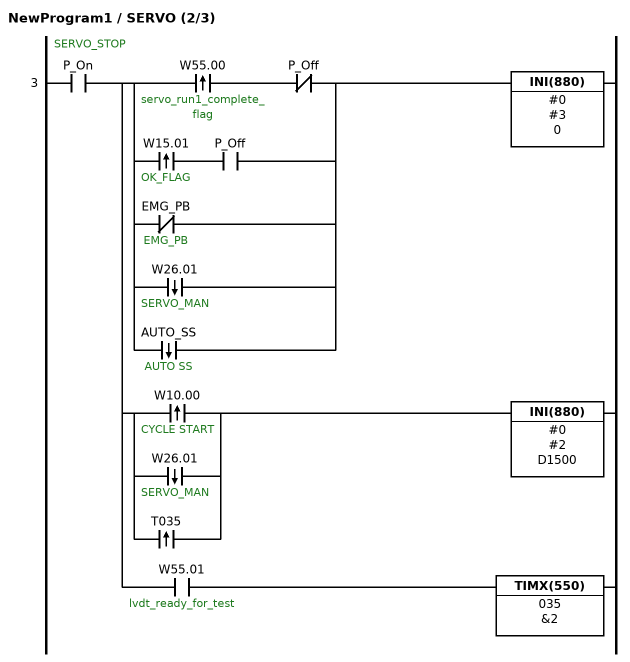
; [picture p24: NewProgram1 / SERVO, rungs 3-3]
; rung 3: SERVO_STOP
LD P_On
OUT TR0
@LD W55.00  ; servo_run1_complete_flag
ANDNOT P_Off
@LD W15.01  ; OK_FLAG
AND P_Off
ORLD
ORNOT EMG_PB  ; EMG_PB
%OR W26.01  ; SERVO_MAN
%OR AUTO_SS  ; AUTO SS
ANDLD
INI(880) #0 #3 0
LD TR0
@LD W10.00  ; CYCLE START
%OR W26.01  ; SERVO_MAN
@OR T035
ANDLD
INI(880) #0 #2 D1500
LD TR0
AND W55.01  ; lvdt_ready_for_test
TIMX(550) 035 &2

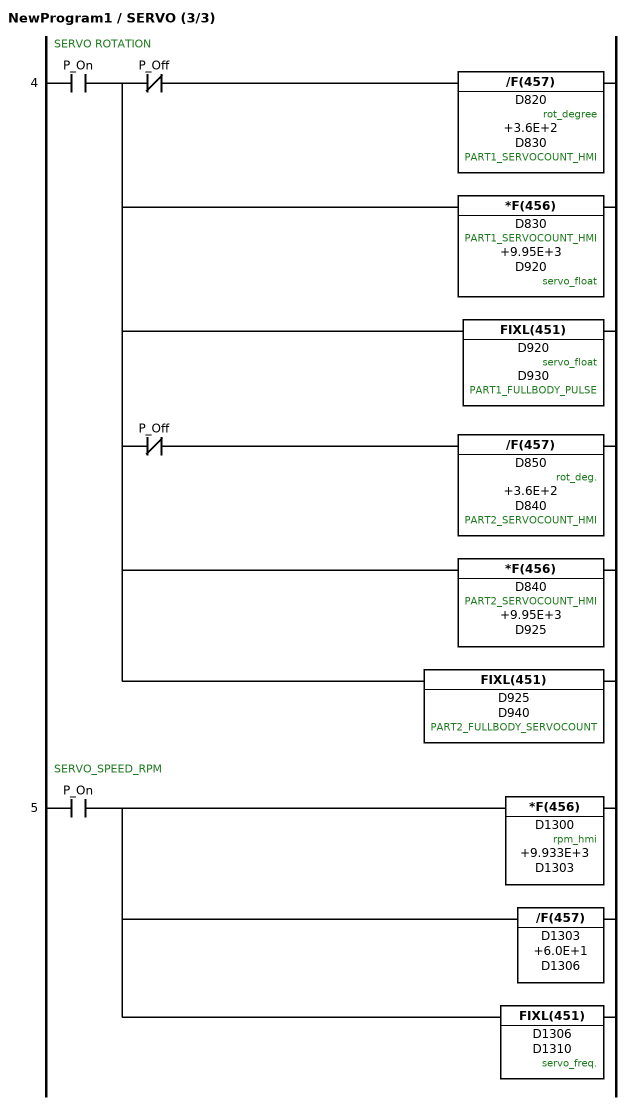
; rung 4: SERVO ROTATION
LD P_On
OUT TR0
ANDNOT P_Off
/F(457) D820 +3.6E+2 D830  ; rot_degree, PART1_SERVOCOUNT_HMI
LD TR0
*F(456) D830 +9.95E+3 D920  ; PART1_SERVOCOUNT_HMI, servo_float
FIXL(451) D920 D930  ; servo_float, PART1_FULLBODY_PULSE
ANDNOT P_Off
/F(457) D850 +3.6E+2 D840  ; rot_deg., PART2_SERVOCOUNT_HMI
LD TR0
*F(456) D840 +9.95E+3 D925  ; PART2_SERVOCOUNT_HMI
FIXL(451) D925 D940  ; PART2_FULLBODY_SERVOCOUNT
; rung 5: SERVO_SPEED_RPM
LD P_On
*F(456) D1300 +9.933E+3 D1303  ; rpm_hmi
/F(457) D1303 +6.0E+1 D1306
FIXL(451) D1306 D1310  ; servo_freq.

### Section MANUAL

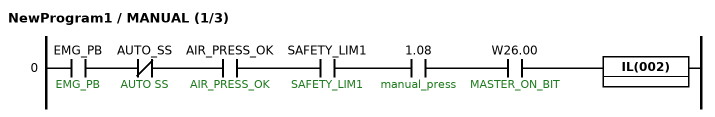
; rung 0
LD EMG_PB  ; EMG_PB
ANDNOT AUTO_SS  ; AUTO SS
AND AIR_PRESS_OK  ; AIR_PRESS_OK
AND SAFETY_LIM1  ; SAFETY_LIM1
AND 1.08  ; manual_press
AND W26.00  ; MASTER_ON_BIT
IL(002)

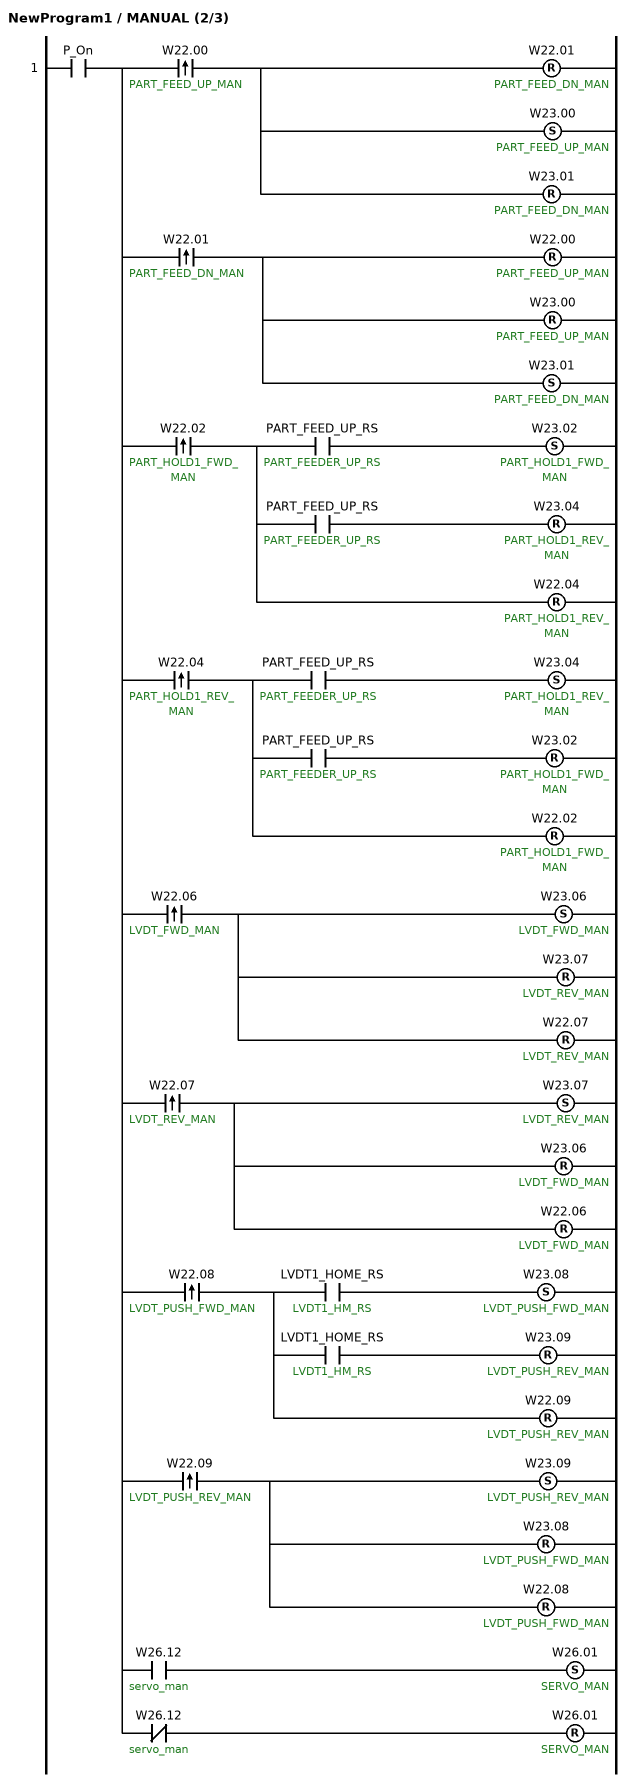
; rung 1
LD P_On
OUT TR0
@AND W22.00  ; PART_FEED_UP_MAN
RSET W22.01  ; PART_FEED_DN_MAN
SET W23.00  ; PART_FEED_UP_MAN
RSET W23.01  ; PART_FEED_DN_MAN
LD TR0
@AND W22.01  ; PART_FEED_DN_MAN
RSET W22.00  ; PART_FEED_UP_MAN
RSET W23.00  ; PART_FEED_UP_MAN
SET W23.01  ; PART_FEED_DN_MAN
LD TR0
@AND W22.02  ; PART_HOLD1_FWD_MAN
OUT TR1
AND PART_FEED_UP_RS  ; PART_FEEDER_UP_RS
SET W23.02  ; PART_HOLD1_FWD_MAN
LD TR1
AND PART_FEED_UP_RS  ; PART_FEEDER_UP_RS
RSET W23.04  ; PART_HOLD1_REV_MAN
LD TR1
RSET W22.04  ; PART_HOLD1_REV_MAN
LD TR0
@AND W22.04  ; PART_HOLD1_REV_MAN
OUT TR1
AND PART_FEED_UP_RS  ; PART_FEEDER_UP_RS
SET W23.04  ; PART_HOLD1_REV_MAN
LD TR1
AND PART_FEED_UP_RS  ; PART_FEEDER_UP_RS
RSET W23.02  ; PART_HOLD1_FWD_MAN
LD TR1
RSET W22.02  ; PART_HOLD1_FWD_MAN
LD TR0
@AND W22.06  ; LVDT_FWD_MAN
SET W23.06  ; LVDT_FWD_MAN
RSET W23.07  ; LVDT_REV_MAN
RSET W22.07  ; LVDT_REV_MAN
LD TR0
@AND W22.07  ; LVDT_REV_MAN
SET W23.07  ; LVDT_REV_MAN
RSET W23.06  ; LVDT_FWD_MAN
RSET W22.06  ; LVDT_FWD_MAN
LD TR0
@AND W22.08  ; LVDT_PUSH_FWD_MAN
OUT TR1
AND LVDT1_HOME_RS  ; LVDT1_HM_RS
SET W23.08  ; LVDT_PUSH_FWD_MAN
LD TR1
AND LVDT1_HOME_RS  ; LVDT1_HM_RS
RSET W23.09  ; LVDT_PUSH_REV_MAN
LD TR1
RSET W22.09  ; LVDT_PUSH_REV_MAN
LD TR0
@AND W22.09  ; LVDT_PUSH_REV_MAN
SET W23.09  ; LVDT_PUSH_REV_MAN
RSET W23.08  ; LVDT_PUSH_FWD_MAN
RSET W22.08  ; LVDT_PUSH_FWD_MAN
LD TR0
AND W26.12  ; servo_man
SET W26.01  ; SERVO_MAN
LD TR0
ANDNOT W26.12  ; servo_man
RSET W26.01  ; SERVO_MAN

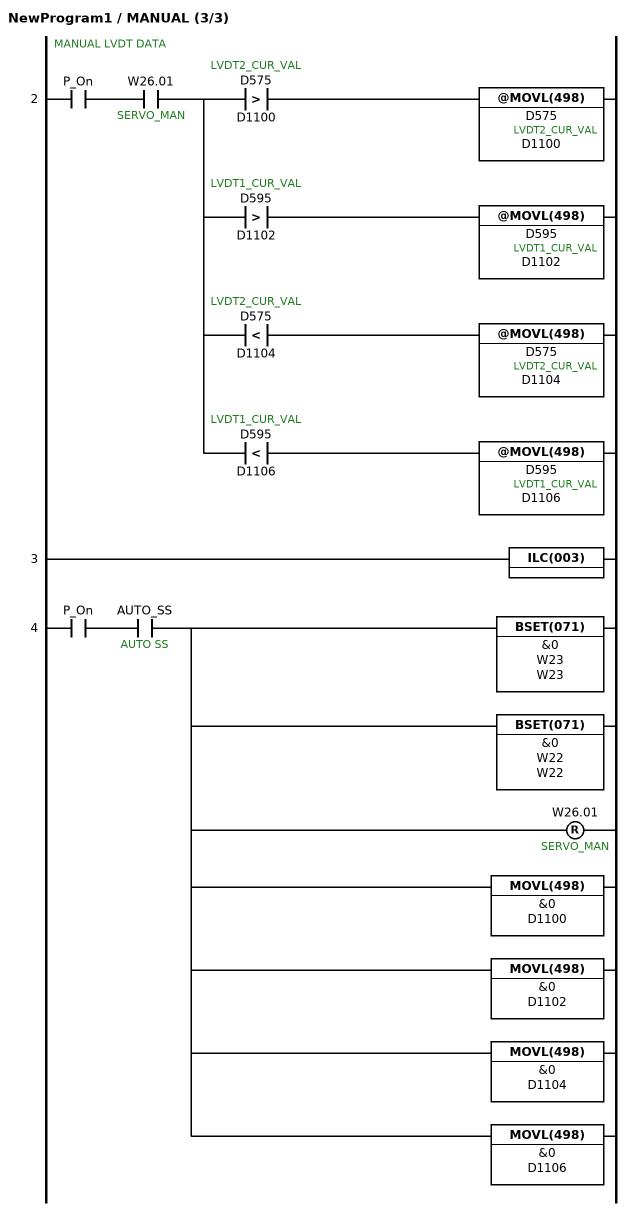
; rung 2: MANUAL LVDT DATA
LD P_On
AND W26.01  ; SERVO_MAN
OUT TR0
AND>F(333) D575 D1100  ; LVDT2_CUR_VAL
@MOVL(498) D575 D1100  ; LVDT2_CUR_VAL
LD TR0
AND>F(333) D595 D1102  ; LVDT1_CUR_VAL
@MOVL(498) D595 D1102  ; LVDT1_CUR_VAL
LD TR0
AND<F(331) D575 D1104  ; LVDT2_CUR_VAL
@MOVL(498) D575 D1104  ; LVDT2_CUR_VAL
LD TR0
AND<F(331) D595 D1106  ; LVDT1_CUR_VAL
@MOVL(498) D595 D1106  ; LVDT1_CUR_VAL
; rung 3
ILC(003)
; rung 4
LD P_On
AND AUTO_SS  ; AUTO SS
BSET(071) &0 W23 W23
BSET(071) &0 W22 W22
RSET W26.01  ; SERVO_MAN
MOVL(498) &0 D1100
MOVL(498) &0 D1102
MOVL(498) &0 D1104
MOVL(498) &0 D1106

### Section DATA_LOG

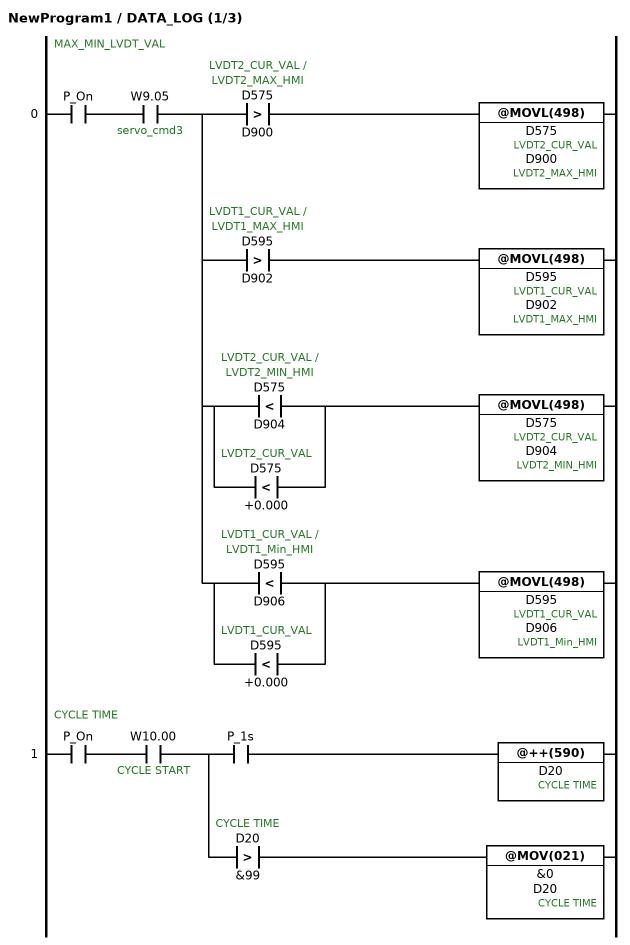
; rung 0: MAX_MIN_LVDT_VAL
LD P_On
AND W9.05  ; servo_cmd3
OUT TR0
AND>F(333) D575 D900  ; LVDT2_CUR_VAL, LVDT2_MAX_HMI
@MOVL(498) D575 D900  ; LVDT2_CUR_VAL, LVDT2_MAX_HMI
LD TR0
AND>F(333) D595 D902  ; LVDT1_CUR_VAL, LVDT1_MAX_HMI
@MOVL(498) D595 D902  ; LVDT1_CUR_VAL, LVDT1_MAX_HMI
LD TR0
LD<F(331) D575 D904  ; LVDT2_CUR_VAL, LVDT2_MIN_HMI
OR<F(331) D575 +0.000  ; LVDT2_CUR_VAL
ANDLD
@MOVL(498) D575 D904  ; LVDT2_CUR_VAL, LVDT2_MIN_HMI
LD TR0
LD<F(331) D595 D906  ; LVDT1_CUR_VAL, LVDT1_Min_HMI
OR<F(331) D595 +0.000  ; LVDT1_CUR_VAL
ANDLD
@MOVL(498) D595 D906  ; LVDT1_CUR_VAL, LVDT1_Min_HMI
; rung 1: CYCLE TIME
LD P_On
AND W10.00  ; CYCLE START
OUT TR0
AND P_1s
@++(590) D20  ; CYCLE TIME
LD TR0
AND>(320) D20 &99  ; CYCLE TIME
@MOV(021) &0 D20  ; CYCLE TIME

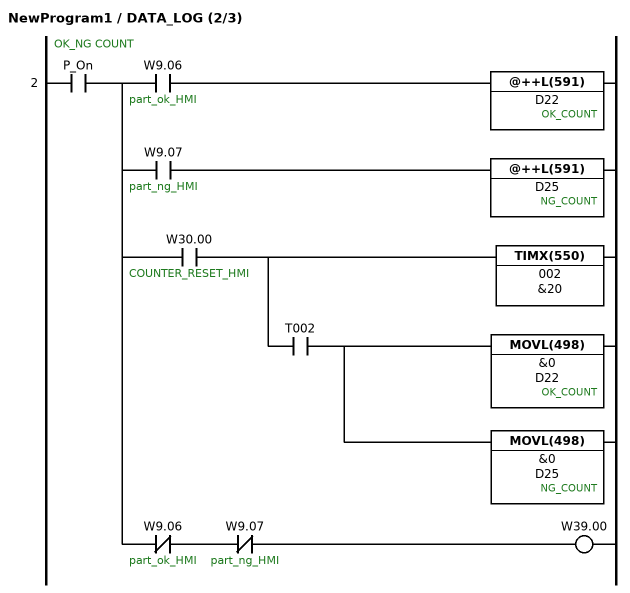
; rung 2: OK_NG COUNT
LD P_On
OUT TR0
AND W9.06  ; part_ok_HMI
@++L(591) D22  ; OK_COUNT
LD TR0
AND W9.07  ; part_ng_HMI
@++L(591) D25  ; NG_COUNT
LD TR0
AND W30.00  ; COUNTER_RESET_HMI
TIMX(550) 002 &20
AND T002
MOVL(498) &0 D22  ; OK_COUNT
MOVL(498) &0 D25  ; NG_COUNT
LD TR0
ANDNOT W9.06  ; part_ok_HMI
ANDNOT W9.07  ; part_ng_HMI
OUT W39.00

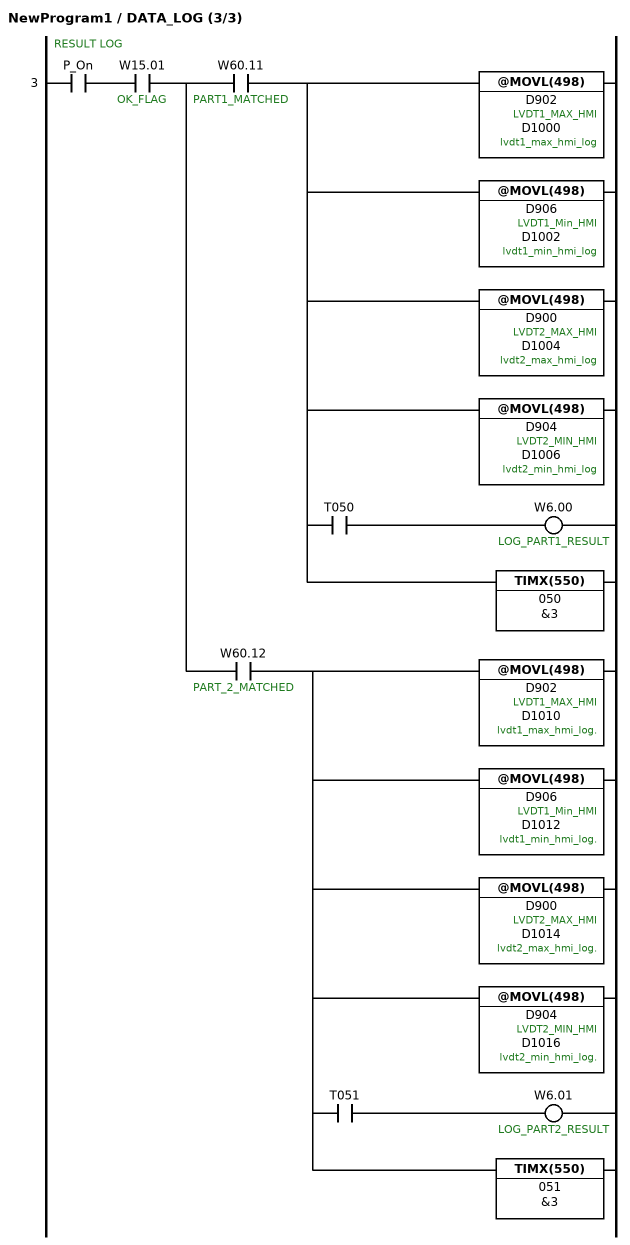
; rung 3: RESULT LOG
LD P_On
AND W15.01  ; OK_FLAG
OUT TR0
AND W60.11  ; PART1_MATCHED
OUT TR1
@MOVL(498) D902 D1000  ; LVDT1_MAX_HMI, lvdt1_max_hmi_log
@MOVL(498) D906 D1002  ; LVDT1_Min_HMI, lvdt1_min_hmi_log
@MOVL(498) D900 D1004  ; LVDT2_MAX_HMI, lvdt2_max_hmi_log
@MOVL(498) D904 D1006  ; LVDT2_MIN_HMI, lvdt2_min_hmi_log
AND T050
OUT W6.00  ; LOG_PART1_RESULT
LD TR1
TIMX(550) 050 &3
LD TR0
AND W60.12  ; PART_2_MATCHED
OUT TR0
@MOVL(498) D902 D1010  ; LVDT1_MAX_HMI, lvdt1_max_hmi_log.
@MOVL(498) D906 D1012  ; LVDT1_Min_HMI, lvdt1_min_hmi_log.
@MOVL(498) D900 D1014  ; LVDT2_MAX_HMI, lvdt2_max_hmi_log.
@MOVL(498) D904 D1016  ; LVDT2_MIN_HMI, lvdt2_min_hmi_log.
AND T051
OUT W6.01  ; LOG_PART2_RESULT
LD TR0
TIMX(550) 051 &3

### Section END
; rung 0
END(001)